FUNCTION_BLOCK ROL (* bitwise rotate left function *)
  (* Standard: 61131-3; Classification: standard bit shift function; Description: Copyright (c) 2013 TU Wien ACIN This program and the accompanying materials are made available under the terms of the Eclipse Public License 2.0 which is available at https://www.eclipse.org/legal/epl-2.0/ SPDX-License-Identifier: EPL-2.0 *)
  (* Version 1.0, 2013-04-22, Monika Wenger, TU Wien ACIN *)
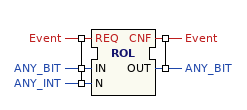
  EVENT_INPUT
    REQ WITH IN, N; (* Service Request *)
  END_EVENT
  EVENT_OUTPUT
    CNF WITH OUT; (* Confirmation of Requested Service *)
  END_EVENT
  VAR_INPUT
    IN : ANY_BIT; (* left-rotated *)
    N : ANY_INT; (* left-rotated by N bits *)
  END_VAR
  VAR_OUTPUT
    OUT : ANY_BIT; (* left-rotated by N zero-filled on right *)
  END_VAR
END_FUNCTION_BLOCK
